Fanuc TP program (LS listing): test2.ls

/PROG  TEST2
/ATTR
OWNER		= MNEDITOR;
COMMENT		= "TEST2";
PROG_SIZE	= 487;
CREATE		= DATE 26-05-05  TIME 16:41:48;
MODIFIED	= DATE 26-05-05  TIME 16:41:48;
FILE_NAME	= TEST2;
VERSION		= 0;
LINE_COUNT	= 1;
MEMORY_SIZE	= 855;
PROTECT		= READ_WRITE;
TCD:  STACK_SIZE	= 0,
      TASK_PRIORITY	= 50,
      TIME_SLICE	= 0,
      BUSY_LAMP_OFF	= 0,
      ABORT_REQUEST	= 0,
      PAUSE_REQUEST	= 0;
DEFAULT_GROUP	= 1,*,*,*,*;
CONTROL_CODE	= 00000000 00000000;
LOCAL_REGISTERS	= 0,0,0;
/APPL
/APPL
/MN
   1:J P[1] 100% CNT100    ;
/POS
P[1]{
   GP1:
	UF : 0, UT : 1,		CONFIG : 'L, 0, 0, 0',
	X =   -22.034000  mm,	Y =  -500.095001  mm,	Z =   227.468002  mm,
	W =  -180.000000 deg,	P =     0.000000 deg,	R =  -148.733994 deg
};
/END
